# EPICS substitutions: db/userHost.substitutions
# Example substitutions file

file "db/dbExample1.db" {
    { user = "hstecherHost" }
}

file db/dbExample2.db {
    pattern { user, no, scan }
        { "hstecherHost", 1, "1 second" }
        { "hstecherHost", 2, "2 second" }
        { "hstecherHost", 3, "5 second" }
}
